% RSLogix 500 project WATER PUMP.RSS, saved by version 8.10.00.18 %
PROJECT "UNTITLED"    % processor: MicroLogix 1500 %

PROGRAM FILES
  LAD 2   6 rungs

DATA FILES
  O0 OUTPUT  4 elements
  I1 INPUT  5 elements
  S2 STATUS  66 elements
  B3 BINARY  1 elements
  T4 TIMER  2 elements
  C5 COUNTER  1 elements
  R6 CONTROL  1 elements
  N7 INTEGER  1 elements
  F8 RESERVED  1 elements

LADDER 2
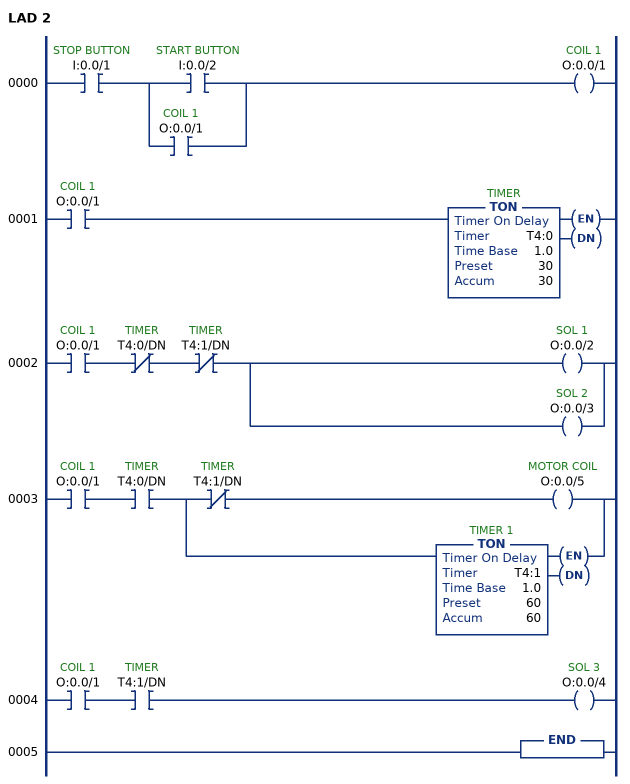
% Rung: 0 %
SOR XIC I:0.0/1 BST XIC I:0.0/2 NXB XIC O:0.0/1 BND OTE O:0.0/1 EOR
%   I:0.0/1  "STOP BUTTON" %
%   I:0.0/2  "START BUTTON" %
%   O:0.0/1  "COIL 1" %
% Rung: 1 %
SOR XIC O:0.0/1 TON T4:0 1.0 30 30 EOR
%   O:0.0/1  "COIL 1" %
%   T4:0  "TIMER" %
% Rung: 2 %
SOR XIC O:0.0/1 XIO T4:0/DN XIO T4:1/DN BST OTE O:0.0/2 NXB OTE O:0.0/3 BND EOR
%   O:0.0/1  "COIL 1" %
%   T4:0/DN  "TIMER" %
%   T4:1/DN  "TIMER" %
%   O:0.0/2  "SOL 1" %
%   O:0.0/3  "SOL 2" %
% Rung: 3 %
SOR XIC O:0.0/1 XIC T4:0/DN BST XIO T4:1/DN OTE O:0.0/5 NXB TON T4:1 1.0 60 60 BND EOR
%   O:0.0/1  "COIL 1" %
%   T4:0/DN  "TIMER" %
%   T4:1/DN  "TIMER" %
%   O:0.0/5  "MOTOR COIL" %
%   T4:1  "TIMER 1" %
% Rung: 4 %
SOR XIC O:0.0/1 XIC T4:1/DN OTE O:0.0/4 EOR
%   O:0.0/1  "COIL 1" %
%   T4:1/DN  "TIMER" %
%   O:0.0/4  "SOL 3" %
% Rung: 5 %
SOR END EOR

REVISION NOTES
  0: XX

DATA TABLE (non-zero values as saved)
DATA T4
% .PRE .ACC %
% T4:0 % 30 30
% T4:1 % 60 60
